FUNCTION_BLOCK FB_ReservoirVolume
VAR_INPUT
	ReservoirVolume : REAL; // L
	ReservoirStartVolume : REAL ; // L
	TotalPipeVolume : REAL ; // L
	PumpFlow : REAL ; // L/s
	
END_VAR
VAR_OUTPUT
	CurrentPipeVolume : REAL ;
END_VAR
VAR
END_VAR

IF (ReservoirVolume <= ReservoirStartVolume) AND (ReservoirVolume >=(ReservoirStartVolume - TotalPipeVolume) ) THEN
	ReservoirVolume := ReservoirVolume - PumpFlow / (1/simulation_parameters.CycleTime) + simulation_parameters.GravityOilFlow/(1/simulation_parameters.CycleTime) ;
	IF ReservoirVolume > ReservoirStartVolume THEN
		ReservoirVolume :=ReservoirStartVolume ;
	ELSIF (ReservoirVolume <= (ReservoirStartVolume - TotalPipeVolume)) THEN
		ReservoirVolume := (ReservoirStartVolume - TotalPipeVolume) ;
	END_IF
ELSIF (ReservoirVolume >= ReservoirStartVolume) THEN
	ReservoirVolume := ReservoirStartVolume - PumpFlow / (1/simulation_parameters.CycleTime);
ELSIF (ReservoirVolume <= (ReservoirStartVolume - TotalPipeVolume)) THEN
	ReservoirVolume := (ReservoirStartVolume - TotalPipeVolume) + simulation_parameters.GravityOilFlow/(1/simulation_parameters.CycleTime) ;
END_IF

IF ReservoirVolume <= ReservoirStartVolume THEN
	CurrentPipeVolume := ReservoirStartVolume - ReservoirVolume ;
END_IF

END_FUNCTION_BLOCK

(* stored: Version 1.1.0.1, ProductVersion 3.1.4024.12
   POU FB_ReservoirVolume: Id {f84219ca-fdc5-4437-ae77-84a5bc33f122}, SpecialFunc None *)
